(* PLC project Generated.project, CODESYS CODESYS V3.5 SP19 Patch 1 *)
(* stored: creationDateTime 2026-09-14T14:47:22.354232, modificationDateTime 2026-09-14T14:47:22.354232 *)

(* ======================================================================= ↔️ ST_TraceTranslation — Trace de blocage terrain de la translation M3 ─────────────────────────────────────────────────────────────── 🎯 Rôle : Publier au technicien « pourquoi la translation M3 ne bouge pas » : permis de mouvement effectif, interlock hauteur, source SafeStop/coupure et cause de blocage priorisée. 📤 Producteur unique : PRG_05_Translation (Data.TranslationTrace). 📥 Consommateur : FB_TroubleshootingView (pure recopie → GVL_Troubleshooting.S_TraceTranslation). 🔒 Lecture seule — aucun calcul de commande n'en dépend. 🕒 BlockReasonTimestamp : ms depuis démarrage PLC (TIME()), latched au dernier changement de BlockReason (1 scan, mémoire). 📄 Doc métier : DOC/AF/AF_Partie-14_Fonction_Troubleshooting/FB_TroubleshootingView_v1.2.md ======================================================================= *)
TYPE ST_TraceTranslation : STRUCT
  MotionPermitEffective : BOOL;  (* Permis de mouvement effectif (agrégat diagnostic : toutes les barrières levées) 🟢 Translation réellement autorisée à se déplacer *)
  EffectivePermitM3_Tremie : BOOL;  (* Permis directionnels par sens (reflet exact des permis appliqués au mouvement M3) 🟢 Permis canonique M3 vers Trémie (reflet lecture seule) *)
  EffectivePermitM3_Maintenance : BOOL;  (* 🟢 Permis canonique M3 vers Maintenance/P1 (reflet lecture seule) *)
  TremieProcessBlockActive : BOOL;  (* 🛑 Approche trémie interdite par process (trémie pleine / grille levée) — recul libre. Motif du permis trémie rouge. *)
  HeightInterlockBlocking : BOOL;  (* 🚧 Interlock hauteur M1/M2 actif (risque collision) *)
  SafeStopActive : BOOL;  (* Source de blocage — pour distinguer l'origine 🟧 SafeStop effectif appliqué (M3_SafeStop_Aggregate) *)
  SafeStopSourceInput : BOOL;  (* 📥 SafeStop issu du module d'entrée (InputModuleFault) *)
  SafeStopSourceSafety : BOOL;  (* 🛡️ SafeStop issu de FB_Safety_Translation (défaut safety) *)
  PowerCutOffActive : BOOL;  (* 🧨 Coupure puissance amont active *)
  DriveOperational : BOOL;  (* 📡 Variateur AC600 opérationnel *)
  FinalInterlockError : BOOL;  (* Barrière finale (frein / redémarrage) 🛑 Défaut barrière finale (frein / redémarrage) *)
  BlockReason : E_TranslationTraceBlockReason;  (* Cause de blocage priorisée + horodatage 🎯 Cause de blocage prioritaire (ordre de priorité croissant) *)
  BlockReasonTimestamp : UDINT;  (* 🕒 ms depuis démarrage PLC (TIME()) — dernier changement de BlockReason *)
END_STRUCT;
END_TYPE

(* values of E_TranslationTraceBlockReason: NONE: ✅ Aucun blocage — permis de mouvement effectif; POWER_CUTOFF: 🧨 Coupure puissance amont (instSafetyTranslationM3.PowerCutOff) — priorité max; SAFESTOP: 🟧 SafeStop effectif (InputModule OR safety M3); SAFETY_FAULT: 🛡️ Défaut safety M3 latched (FB_Safety_Translation.Fault.Error); HEIGHT_INTERLOCK: 🚧 Interlock hauteur M1/M2 actif (risque collision); DRIVE_UNAVAILABLE: 📡 Variateur AC600 injoignable / non opérationnel; FINAL_INTERLOCK: 🛑 Barrière finale en défaut (frein / redémarrage); FAULT: ❌ Défaut mouvement M3 latched (FB_Translation.Fault.Error) *)

{attribute 'qualified_only'}
{attribute 'strict'}
TYPE E_TranslationTraceBlockReason : (NONE := 0, POWER_CUTOFF := 1, SAFESTOP := 2, SAFETY_FAULT := 3, HEIGHT_INTERLOCK := 4, DRIVE_UNAVAILABLE := 5, FINAL_INTERLOCK := 6, FAULT := 7);
END_TYPE
